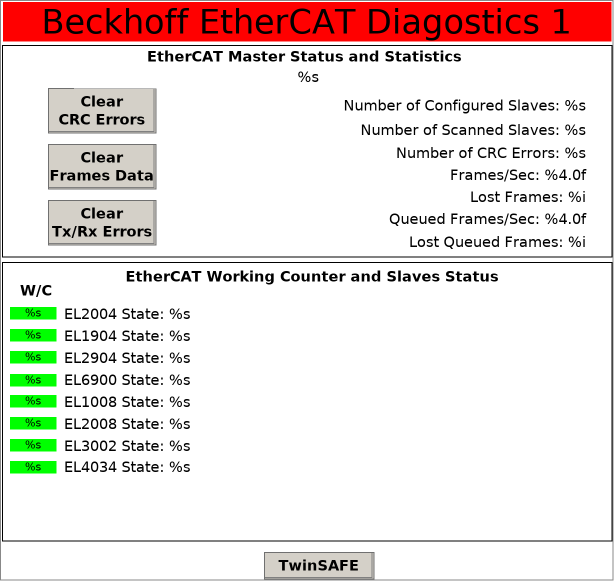
VISUALIZATION EtherCAT_Diag1  // 614x581
    Button (264,552 110x27), "TwinSAFE"
        OnMouseClick: change screen: TwinSAFE
    RoundedRectangle (3,2 608x39), "Beckhoff EtherCAT Diagostics 1"
    RoundedRectangle (2,45 610x212)
    RoundedRectangle (2,262 610x279)
    Label (152,45 305x23), "EtherCAT Master Status and Statistics"
    Button (48,88 108x45), "Clear CRC Errors"
        tap g_xHMI_CearMFStatCRCs
    Label (123,265 378x23), "EtherCAT Working Counter and Slaves Status"
    Button (48,144 108x45), "Clear Frames Data"
        tap g_xHMI_ClearMFStatFrames
    Button (48,200 108x45), "Clear Tx/Rx Errors"
        tap g_xHMI_ClearMFStatTxRxErr
    Label (14,279 44x23), "W/C"
    Rectangle (74,66 469x22), "%s", text variable: g_sHMI_StateMaster
    Rectangle (323,97 266x17), "Number of Configured Slaves: %s", text variable: g_uiHMI_ConfSlaves
    Rectangle (327,121 262x18), "Number of Scanned Slaves: %s", text variable: g_uiHMI_ScannedSlaves
    Rectangle (326,144 263x18), "Number of CRC Errors: %s", text variable: g_dwHMI_TotalCrcErrors
    Rectangle (321,166 268x18), "Frames/Sec: %4.0f", text variable: g_lrHMI_FramesPerSecond
    Rectangle (323,188 266x18), "Lost Frames: %i", text variable: g_udiHMI_LostFrames
    Rectangle (324,210 265x18), "Queued Frames/Sec: %4.0f", text variable: g_lrHMI_QueuedFramesPerSecond
    Rectangle (325,233 264x18), "Lost Queued Frames: %i", text variable: g_udiHMI_LostQueuedFrames
    Rectangle (61,303 520x22), "EL2004 State: %s", text variable: g_sHMI_StateEL2004
    Rectangle (61,325 520x22), "EL1904 State: %s", text variable: g_sHMI_StateEL1904
    Rectangle (61,347 520x22), "EL2904 State: %s", text variable: g_sHMI_StateEL2904
    Rectangle (61,369 520x22), "EL6900 State: %s", text variable: g_sHMI_StateEL6900
    Rectangle (61,391 520x22), "EL1008 State: %s", text variable: g_sHMI_StateEL1008
    Rectangle (61,413 520x22), "EL2008 State: %s", text variable: g_sHMI_StateEL2008
    Rectangle (61,435 520x22), "EL3002 State: %s", text variable: g_sHMI_StateEL3002
    Rectangle (61,456 520x22), "EL4034 State: %s", text variable: g_sHMI_StateEL4034
    Rectangle (10,307 46x12), "%s", text variable: g_xEL2004_Wc
    Rectangle (10,329 46x12), "%s", text variable: g_xEL1904_Wc
    Rectangle (10,351 46x12), "%s", text variable: g_xEL2904_Wc
    Rectangle (10,374 46x12), "%s", text variable: g_xEL6900_Wc
    Rectangle (10,395 46x12), "%s", text variable: g_xEL1008_Wc
    Rectangle (10,417 46x12), "%s", text variable: g_xEL2008_Wc
    Rectangle (10,439 46x12), "%s", text variable: g_xEL3002_Wc
    Rectangle (10,461 46x12), "%s", text variable: g_xEL4034_Wc
END_VISUALIZATION

(* stored: Version 1.1.0.1, ProductVersion 3.1.0.18
   Visu EtherCAT_Diag1: Id {e106253d-815d-4bb5-9cde-fb194eb0b815} *)
